# B&R Automation Studio project Kesim (part 5)

### CsvHandling.typ - Package data types
```iecst
(********************************************************************
 * COPYRIGHT -- Bernecker + Rainer
 ********************************************************************
 * Package: CSVHandling
 * File: CSVHandling.typ
 * Author: blanca-gutim
 * Created: December 04, 2012
 ********************************************************************
 * Data types of package CSVHandling
 ********************************************************************)
(**)
(*Enumeration to manage the state machine states*)

TYPE
	emu_CSVControl_State :
		(
		C_MS_CSV_FILE_HAND_INIT := 0, (*Init state*)
		C_MS_CSV_FILE_HAND_WAIT_CMD, (*Wait commad state -Standstill state*)
		C_MS_CSV_FILE_HAND_READ, (*Read CSV file state*)
		C_MS_CSV_FILE_HAND_GEN_FILE_NAME, (*Generate file name state*)
		C_MS_CSV_FILE_HAND_SEARCH_FILE, (*Search for the specified file name*)
		C_MS_CSV_FILE_HAND_WAIT_OVRW_OK, (*Wait overwrite confirmation state*)
		C_MS_CSV_FILE_HAND_SEARCH_VAR, (*Search the variables that are part of the CSV file state*)
		C_MS_CSV_FILE_HAND_WRITE, (*Write CSV file state*)
		C_MS_CSV_FILE_HAND_ERROR, (*General error state*)
		C_MS_CSV_FILE_HAND_ACK_ERROR, (*Acknowledge error state*)
		C_MS_CSV_FILE_HAND_NOERROR (*Error State - No error*)
		);
END_TYPE

(**)
(*========================================================================================================*)
(*CSV control interface type*)
(*========================================================================================================*)

TYPE
	CSV_Ctrl_typ : 	STRUCT
		In : CSV_Ctrl_In_typ; (*Inputs*)
		Out : CSV_Ctrl_Out_typ; (*Outputs*)
	END_STRUCT;
END_TYPE

(*========================================================================================================*)
(*CSV control: input sub-interface type*)
(*========================================================================================================*)

TYPE
	CSV_Ctrl_In_typ : 	STRUCT
		Cmd : CSV_Ctrl_In_Cmd_typ; (*Input commands*)
		Par : CSV_Ctrl_In_Par_typ; (*Input parameters *)
		Stat : CSV_Ctrl_In_Stat_typ; (*Input status*)
	END_STRUCT;
END_TYPE

(*CSV control: input commands sub-interface type*)

TYPE
	CSV_Ctrl_In_Cmd_typ : 	STRUCT
		ReadFile : BOOL; (*Read file command*)
		WriteFile : BOOL; (*Write file command*)
		OverwriteFile : BOOL; (*Overwrite file command*)
		NotOverwriteFile : BOOL; (*Do not overwrite file command*)
		ErrorAcknowledge : BOOL; (*Acknowledge error command*)
	END_STRUCT;
END_TYPE

(*CSV control: input parameters sub-interface type*)

TYPE
	CSV_Ctrl_In_Par_typ : 	STRUCT
		FileDeviceName : STRING[50]; (*File Device name*)
		FileName : STRING[255]; (*File name*)
		Path : STRING[255]; (*Path to the file*)
		Header : CSV_Ctrl_In_Par_Header_typ; (*Header input parameters substructure*)
	END_STRUCT;
END_TYPE

(*Header input parameters substructure*)

TYPE
	CSV_Ctrl_In_Par_Header_typ : 	STRUCT
		Enable : BOOL; (*Enable header in CSV file*)
		MachineNr : STRING[80]; (*Machine number*)
		Comment : STRING[80]; (*Header comment*)
		Version : STRING[80]; (*Version*)
	END_STRUCT;
END_TYPE

(*CSV control: input status sub-interface type*)

TYPE
	CSV_Ctrl_In_Stat_typ : 	STRUCT
		NOT_USED : BOOL;
	END_STRUCT;
END_TYPE

(*========================================================================================================*)
(*CSV control: output sub-interface type*)
(*========================================================================================================*)

TYPE
	CSV_Ctrl_Out_typ : 	STRUCT
		Cmd : CSV_Ctrl_Out_Cmd_typ; (*Output commands*)
		Par : CSV_Ctrl_Out_Par_typ; (*Output parameters *)
		Stat : CSV_Ctrl_Out_Stat_typ; (*Output status*)
	END_STRUCT;
END_TYPE

(*CSV control: output commands sub-interface type*)

TYPE
	CSV_Ctrl_Out_Cmd_typ : 	STRUCT
		NOT_USED : BOOL;
	END_STRUCT;
END_TYPE

(*CSV control: output parameters sub-interface type*)

TYPE
	CSV_Ctrl_Out_Par_typ : 	STRUCT
		NOT_USED : BOOL;
	END_STRUCT;
END_TYPE

(*CSV control: output status sub-interface type*)

TYPE
	CSV_Ctrl_Out_Stat_typ : 	STRUCT
		MainState : DINT; (*Main state in numeric format*)
		MainState_Text : STRING[32]; (*Main state in text format*)
		VariableNames : ARRAY[0..C_NR_VARIABLES_CSVFILE_MINUS1]OF STRING[30]; (*Names of the variables that are part of the CSV file*)
		CmdDone : CSV_Ctrl_In_Cmd_typ; (*Command done*)
		FileAlreadyExists : BOOL; (*Flag to show that the CSV file already exists (in write process)*)
		ReadyForCmd : BOOL; (*Variable to show that the program is ready to get a new command*)
(*		Error : Error_Type; (*Error information*)
	END_STRUCT;
END_TYPE
```

### CsvHandling.var - Package variables
```iecst
(********************************************************************
 * COPYRIGHT -- Bernecker + Rainer
 ********************************************************************
 * Package: RecipeHandling
 * File: CsvHandling.var
 * Author: blanca-gutim
 * Created: December 04, 2012
 ********************************************************************
 * Variables of package RecipeHandling
 ********************************************************************)
(**)
(*========================================================================================================*)
(*Program variables*)
(*========================================================================================================*)
VAR
	gCSV_Ctrl : CSV_Ctrl_typ; (*CSV control interface*)
END_VAR
```

### Program Logical/CuttingTable/RecipeHandling/CsvHandling/CSV_Ctrl (IEC) - CSV file control program

#### CSV_CtrlCyclic.st - Cyclic code
```iecst
(********************************************************************
 * COPYRIGHT -- Bernecker + Rainer
 ********************************************************************
 * PROGRAM: gCSV_Ctrl
 * File: gCSV_CtrlCyclic.st
 * Author: blanca-gutim
 * Created: December 06, 2012
 ********************************************************************
 * Implementation OF PROGRAM gCSV_Ctrl
 ********************************************************************)

PROGRAM _CYCLIC

	//Update inputs
	Action_Input;

	//====================================================================================================
	//
	//									MAIN STATE MACHINE
	//
	//====================================================================================================
	IF TON_Init.Q THEN
		TON_Init.IN := FALSE;
		//FUB execution
		Init_CSVHandling();

		//Check if the FUB is done
		IF (Init_CSVHandling.status = ERR_FUB_BUSY) THEN
			//The FUB is busy
		ELSE
			IF (Init_CSVHandling.status = ERR_OK) THEN
				//FUB executed successfully
			ELSE
				//Error -> Save information about error
				gCSV_Ctrl.Out.Stat.Error.Number		:= Init_CSVHandling.status;
				gCSV_Ctrl.Out.Stat.Error.Text.Line1	:= TaskName;
				gCSV_Ctrl.Out.Stat.Error.Text.Line2	:= StateStrings[MainState];
				ErrorState							:= MainState;
				MainState							:= C_MS_CSV_FILE_HAND_ERROR;
			END_IF
		END_IF
	END_IF;
	CASE MainState OF

		//============================================================================================
		C_MS_CSV_FILE_HAND_INIT:					//INITIALIZATION STATE
			//============================================================================================

			//Initialization done -> Go to Wait Command state
			MainState 			:= C_MS_CSV_FILE_HAND_WAIT_CMD;

		//============================================================================================
		C_MS_CSV_FILE_HAND_WAIT_CMD:				//STANDSTILL STATE
			//============================================================================================

			//WAIT FOR COMMANDS
			IF (gCSV_Ctrl.Out.Stat.ReadyForCmd = TRUE) THEN
				IF (gCSV_Ctrl.In.Cmd.ReadFile > OldInputs.Cmd.ReadFile) THEN
					//Go to Read CSV file state
					MainState			:= C_MS_CSV_FILE_HAND_READ;
				ELSIF (gCSV_Ctrl.In.Cmd.WriteFile > OldInputs.Cmd.WriteFile) THEN
					//Go to the first state when a file is written
					MainState			:= C_MS_CSV_FILE_HAND_SEARCH_FILE;
				ELSE
					//Stay in Wait Command state
					MainState 			:= C_MS_CSV_FILE_HAND_WAIT_CMD;
				END_IF
			END_IF

			//Update the output ReadyForCmd
			IF (MainState = C_MS_CSV_FILE_HAND_WAIT_CMD) THEN
				gCSV_Ctrl.Out.Stat.ReadyForCmd	:= TRUE;
			ELSE
				gCSV_Ctrl.Out.Stat.ReadyForCmd	:= FALSE;
			END_IF

		//============================================================================================
		C_MS_CSV_FILE_HAND_READ:				//READ CSV FILE
			//============================================================================================

			//FUB parameters
			ReadFile_CSVHandling.pDevice			:= ADR(gCSV_Ctrl.In.Par.FileDeviceName);
			ReadFile_CSVHandling.pPath				:= ADR(gCSV_Ctrl.In.Par.Path);
			ReadFile_CSVHandling.pFileName			:= ADR(gCSV_Ctrl.In.Par.FileName);
			ReadFile_CSVHandling.Separator			:= C_SEPARATOR;	//Check constant to see the ASCII code of the actual separator
			ReadFile_CSVHandling.No_DatatypControl	:= 1;
			ReadFile_CSVHandling.IgnoreError		:= 1;
			ReadFile_CSVHandling.Options			:= 0;

			//FUB execution
			ReadFile_CSVHandling();

			//Chec if the FUB is done
			IF (ReadFile_CSVHandling.status = ERR_FUB_BUSY) THEN
				//The FUB is busy
			ELSE
				IF (ReadFile_CSVHandling.status = ERR_OK) THEN
					//FUB executed successfully -> Go to wait command state
					MainState							:= C_MS_CSV_FILE_HAND_WAIT_CMD;
					//Set output status command done
					gCSV_Ctrl.Out.Stat.CmdDone.ReadFile	:= TRUE;
				ELSE
					//Error -> Save information about error
					gCSV_Ctrl.Out.Stat.Error.Number		:= ReadFile_CSVHandling.status;
					gCSV_Ctrl.Out.Stat.Error.Text.Line1	:= TaskName;
					gCSV_Ctrl.Out.Stat.Error.Text.Line2	:= StateStrings[MainState];
					ErrorState							:= MainState;
					MainState							:= C_MS_CSV_FILE_HAND_ERROR;
				END_IF
			END_IF

		//============================================================================================
		C_MS_CSV_FILE_HAND_SEARCH_FILE:				//SEARCH FOR THE SPECIFIED FILE NAME
			//============================================================================================

			//FUB parameters
			ToSearchFileName						:= gCSV_Ctrl.In.Par.Path;
			strcat(ADR(ToSearchFileName), ADR(gCSV_Ctrl.In.Par.FileName));
			SearchFileName_CSVHandling.pFileName	:= ADR(ToSearchFileName);
			SearchFileName_CSVHandling.pDevice		:= ADR(gCSV_Ctrl.In.Par.FileDeviceName);

			//FUB execution
			SearchFileName_CSVHandling();

			//Chec if the FUB is done
			IF (SearchFileName_CSVHandling.status = ERR_FUB_BUSY) THEN
				//The FUB is busy
			ELSE
				IF (SearchFileName_CSVHandling.status = FILE_NOT_FOUND) THEN
					//FUB executed successfully, and the file does not exist -> Go to search variables that are part of the CSV file
					MainState							:= C_MS_CSV_FILE_HAND_SEARCH_VAR;
				ELSIF  (SearchFileName_CSVHandling.status = FILE_FOUND) THEN
					//FUB executed successfully, the file already exists -> Set flag to show this state, wait for confirmation to overwrite the file
					gCSV_Ctrl.Out.Stat.FileAlreadyExists := TRUE;
					MainState							:= C_MS_CSV_FILE_HAND_WAIT_OVRW_OK;
				ELSE
					//Error -> Save information about error
					gCSV_Ctrl.Out.Stat.Error.Number		:= SearchFileName_CSVHandling.status;
					gCSV_Ctrl.Out.Stat.Error.Text.Line1	:= TaskName;
					gCSV_Ctrl.Out.Stat.Error.Text.Line2	:= StateStrings[MainState];
					ErrorState							:= MainState;
					MainState							:= C_MS_CSV_FILE_HAND_ERROR;
				END_IF
			END_IF

		//============================================================================================
		C_MS_CSV_FILE_HAND_WAIT_OVRW_OK:			//WAIT FOR USER CONFIRMATION TO OVERWRITE THE FILE
			//============================================================================================

			//Wait for an user command about the possibility of overwriting the file
			IF (gCSV_Ctrl.In.Cmd.OverwriteFile > OldInputs.Cmd.OverwriteFile) THEN
				//Reset flag and go to search variables that are part of the CSV file
				gCSV_Ctrl.Out.Stat.FileAlreadyExists 		:= FALSE;
				MainState									:= C_MS_CSV_FILE_HAND_SEARCH_VAR;
			ELSIF (gCSV_Ctrl.In.Cmd.NotOverwriteFile > OldInputs.Cmd.NotOverwriteFile) THEN
				//Set output status commands done, flag and go to wait command
				gCSV_Ctrl.Out.Stat.CmdDone.WriteFile			:= TRUE;
				gCSV_Ctrl.Out.Stat.CmdDone.NotOverwriteFile	:= TRUE;
				gCSV_Ctrl.Out.Stat.FileAlreadyExists 		:= FALSE;
				MainState									:= C_MS_CSV_FILE_HAND_WAIT_CMD;
			END_IF

		//============================================================================================
		C_MS_CSV_FILE_HAND_SEARCH_VAR:				//SEARCH VARIABLES THAT ARE PART OF THE CSV FILE
			//============================================================================================

			//FUB parameters
			Search_CSVHandling.pStructName		:= Init_CSVHandling.pStructName;
			Search_CSVHandling.NumOfStructs		:= Init_CSVHandling.NumOfStructs;
			Search_CSVHandling.pStructMem		:= Init_CSVHandling.pStructMem;
			Search_CSVHandling.MemLen			:= Init_CSVHandling.MemCounter;
			Search_CSVHandling.Options			:= 0;
			Search_CSVHandling.FullNameLenght	:= C_SHOW_VAR_NAME_OPTION;
			Search_CSVHandling.FileHeader		:= gCSV_Ctrl.In.Par.Header.Enable;
			Search_CSVHandling.Separator		:= C_SEPARATOR; //Check constants to see the ASCII code
			Search_CSVHandling.pMaschineNo		:= ADR(gCSV_Ctrl.In.Par.Header.MachineNr);
			Search_CSVHandling.pComment			:= ADR(gCSV_Ctrl.In.Par.Header.Comment);
			Search_CSVHandling.pVersion			:= ADR(gCSV_Ctrl.In.Par.Header.Version);

			//FUB execution
			Search_CSVHandling;

			//Chec if the FUB is done
			IF (Search_CSVHandling.status = ERR_FUB_BUSY) THEN
				//The FUB is busy
			ELSE
				IF (Search_CSVHandling.status = ERR_OK) THEN
					//FUB executed successfully -> Go to write CSV file
					MainState							:= C_MS_CSV_FILE_HAND_WRITE;
				ELSE
					//Error -> Save information about error
					gCSV_Ctrl.Out.Stat.Error.Number		:= Search_CSVHandling.status;
					gCSV_Ctrl.Out.Stat.Error.Text.Line1	:= TaskName;
					gCSV_Ctrl.Out.Stat.Error.Text.Line2	:= StateStrings[MainState];
					ErrorState							:= MainState;
					MainState							:= C_MS_CSV_FILE_HAND_ERROR;
				END_IF
			END_IF

		//============================================================================================
		C_MS_CSV_FILE_HAND_WRITE:				//WRITE THE CSV FILE
			//============================================================================================

			//FUB parameters
			WriteFile_CSVHandling.pFileName		:= ADR(gCSV_Ctrl.In.Par.FileName);
			WriteFile_CSVHandling.pDevice		:= ADR(gCSV_Ctrl.In.Par.FileDeviceName);
			WriteFile_CSVHandling.pPath			:= ADR(gCSV_Ctrl.In.Par.Path);
			WriteFile_CSVHandling.pStructMem	:= Init_CSVHandling.pStructMem;
			WriteFile_CSVHandling.MemLen		:= Search_CSVHandling.FileLen;
			WriteFile_CSVHandling.Mode			:= FILE_OW;

			//FUB execution
			WriteFile_CSVHandling;

			//Chec if the FUB is done
			IF (WriteFile_CSVHandling.status = ERR_FUB_BUSY) THEN
				//The FUB is busy
			ELSE
				IF (WriteFile_CSVHandling.status = ERR_OK) THEN
					//FUB executed successfully -> Go to wait command
					MainState									:= C_MS_CSV_FILE_HAND_WAIT_CMD;
					//Set output status command done
					gCSV_Ctrl.Out.Stat.CmdDone.WriteFile			:= TRUE;
					IF (gCSV_Ctrl.In.Cmd.OverwriteFile = TRUE) THEN
						gCSV_Ctrl.Out.Stat.CmdDone.OverwriteFile	:= TRUE;
					END_IF
				ELSE
					//Error -> Save information about error
					gCSV_Ctrl.Out.Stat.Error.Number				:= WriteFile_CSVHandling.status;
					gCSV_Ctrl.Out.Stat.Error.Text.Line1			:= TaskName;
					gCSV_Ctrl.Out.Stat.Error.Text.Line2			:= StateStrings[MainState];
					ErrorState									:= MainState;
					MainState									:= C_MS_CSV_FILE_HAND_ERROR;
				END_IF
			END_IF

		//============================================================================================
		C_MS_CSV_FILE_HAND_ERROR:				//ERROR HANDLING
			//============================================================================================

			//Wait for user acknowledge
			IF (gCSV_Ctrl.In.Cmd.ErrorAcknowledge > OldInputs.Cmd.ErrorAcknowledge) THEN
				//The user wants to acknowledge the error -> Next step: Go to Acknowledge Error State
				MainState 				:= C_MS_CSV_FILE_HAND_ACK_ERROR;
			END_IF

		//============================================================================================
		C_MS_CSV_FILE_HAND_ACK_ERROR:			//ACKNOWLEDGE ERROR
			//============================================================================================

			//Clear error information
			gCSV_Ctrl.Out.Stat.Error.Number				:= 0;
			memset(ADR(gCSV_Ctrl.Out.Stat.Error.Text), 0, SIZEOF(gCSV_Ctrl.Out.Stat.Error.Text));
			ErrorState									:= C_MS_CSV_FILE_HAND_NOERROR;
			MainState									:= C_MS_CSV_FILE_HAND_WAIT_CMD;
			//Error acknowledged
			gCSV_Ctrl.Out.Stat.CmdDone.ErrorAcknowledge	:= TRUE;
			//Acknowledge done -> Next step: Go to Init State
			MainState 									:= C_MS_CSV_FILE_HAND_INIT;

		ELSE

			//============================================================================================

			//The program sould not come here
			MainState 								:= C_MS_CSV_FILE_HAND_ERROR;
			gCSV_Ctrl.Out.Stat.Error.Number			:= 0;
			gCSV_Ctrl.Out.Stat.Error.Text.Line1		:= TaskName;
			gCSV_Ctrl.Out.Stat.Error.Text.Line2		:= 'Not defined state in state machine';
			ErrorState								:= MainState;
			MainState								:= C_MS_CSV_FILE_HAND_ERROR;

			//============================================================================================

	END_CASE

	TON_Init();
	//Update old inputs variable
	OldInputs	:= gCSV_Ctrl.In;

	//Update outputs
	Action_Output;

END_PROGRAM
```

#### CSV_CtrlInit.st - Initialization code
```iecst
(********************************************************************
 * COPYRIGHT -- Bernecker + Rainer
 ********************************************************************
 * Program: gCSV_Ctrl
 * File: gCSV_CtrlInit.st
 * Author: blanca-gutim
 * Created: December 06, 2012
 ********************************************************************
 * Implementation of program gCSV_Ctrl
 ********************************************************************)

PROGRAM _INIT

	//Init of task name
	TaskName	:= 'CSV_Ctrl';

	//Init of variable to get state names in text format
	StateStrings[C_MS_CSV_FILE_HAND_INIT]			:= 'C_MS_CSV_FILE_HAND_INIT';
	StateStrings[C_MS_CSV_FILE_HAND_WAIT_CMD]		:= 'C_MS_CSV_FILE_HAND_WAIT_CMD';
	StateStrings[C_MS_CSV_FILE_HAND_READ]			:= 'C_MS_CSV_FILE_HAND_READ';
	StateStrings[C_MS_CSV_FILE_HAND_GEN_FILE_NAME]	:= 'C_MS_CSV_FILE_HAND_GEN_FILE_NAME';
	StateStrings[C_MS_CSV_FILE_HAND_SEARCH_FILE]	:= 'C_MS_CSV_FILE_HAND_SEARCH_FILE';
	StateStrings[C_MS_CSV_FILE_HAND_WAIT_OVRW_OK]	:= 'C_MS_CSV_FILE_HAND_WAIT_OVRW_OK';
	StateStrings[C_MS_CSV_FILE_HAND_SEARCH_VAR]		:= 'C_MS_CSV_FILE_HAND_SEARCH_VAR';
	StateStrings[C_MS_CSV_FILE_HAND_WRITE]			:= 'C_MS_CSV_FILE_HAND_WRITE';
	StateStrings[C_MS_CSV_FILE_HAND_ERROR]			:= 'C_MS_CSV_FILE_HAND_ERROR';
	StateStrings[C_MS_CSV_FILE_HAND_ACK_ERROR]		:= 'C_MS_CSV_FILE_HAND_ACK_ERROR';
	StateStrings[C_MS_CSV_FILE_HAND_NOERROR]		:= 'C_MS_CSV_FILE_HAND_NOERROR';

	//****************************************************************************************************************
	//****************************************************************************************************************
	//THIS PART OF THE CODE MUST BE CONFIGURED FOR EACH APPLICATION
	//CHECK THE VALUE OF THE CONSTANT: C_NR_VARIABLES_CSVFILE_MINUS_1
	//DELETE THE VARIABLES AND STRUCTURES FOR TESTING: TestVar1 AND TestVar2
	//****************************************************************************************************************
	//****************************************************************************************************************
	//Init of the variables that are going to take part in the CSV file
	//Addresses of the names of the variables
	pVarNames[0] 	:= ADR('gParameters');
	//Sizes of the variables
	VarSizes[0]		:= SIZEOF(gParameters);
	//Show output information about the involved variables
	gCSV_Ctrl.Out.Stat.VariableNames[0] := 'gParameters';
	//****************************************************************************************************************
	//****************************************************************************************************************

	//Init of machine state and error information
	MainState 	:= C_MS_CSV_FILE_HAND_INIT;
	ErrorState	:= C_MS_CSV_FILE_HAND_NOERROR;

	//================================================================================================================
	//Calculate the necessary size of the memory to save the CSV-file on the compact flash and allocate the memory
	//================================================================================================================

	//FUB parameters
	Init_CSVHandling.pStructName	:= ADR(pVarNames);
	Init_CSVHandling.NumOfStructs	:= C_NR_VARIABLES_CSVFILE_MINUS1 + 1;
	Init_CSVHandling.FullNameLenght	:= C_SHOW_VAR_NAME_OPTION;
	Init_CSVHandling.Options		:= 0;

	TON_Init.PT := T#5S;
	TON_Init.IN := TRUE;

END_PROGRAM
```

#### CSV_Ctrl.var - Local variables
```iecst
(********************************************************************
 * COPYRIGHT -- Bernecker + Rainer
 ********************************************************************
 * Program: CSV_Ctrl
 * File: CSV_Ctrl.var
 * Author: blanca-gutim
 * Created: December 06, 2012
 ********************************************************************
 * Local variables of program CSV_Ctrl
 ********************************************************************)
(**)
(*================================================
Program variables
================================================*)
VAR
	TaskName : STRING[20]; (*Name of the actual task, used for error handling*)
	MainState : emu_CSVControl_State; (*Main state for the control of the state machine*)
	ErrorState : emu_CSVControl_State; (*Variable used to identify in wich state an error occurs*)
	OldInputs : CSV_Ctrl_In_typ; (*Variable used to detect edges in the inputs*)
	StateStrings : ARRAY[0..15] OF STRING[32]; (*Array with the names of the possible states (update if the number of states is increased)*)
	pVarNames : ARRAY[0..C_NR_VARIABLES_CSVFILE_MINUS1] OF UDINT; (*Addresses of the variables that are part of the CSV file*)
	VarSizes : ARRAY[0..C_NR_VARIABLES_CSVFILE_MINUS1] OF UDINT; (*Sizes of the variables that are part of the CSV file*)
	ToSearchFileName : STRING[255] := ''; (*File name to search by the FUB*)
END_VAR
(**)
(*================================================*)
(*Constants*)
(*================================================*)
(**)
(**)
(*===========================================================================================================================================================*)
(*FUB´S DECLARATION*)
(*===========================================================================================================================================================*)
VAR
	Init_CSVHandling : CSV_Init; (*Calculate the necessary size of the memory to save the CSV-file on the compact flash and allocate the memory*)
	ReadFile_CSVHandling : CSV_ReadFile; (*Read a CSV-file*)
	Search_CSVHandling : CSV_Search; (*Search the specified variable (structure) and create the completed CSV_File entries in the RAM*)
	SearchFileName_CSVHandling : SearchFileName; (*Searching for a file name*)
	WriteFile_CSVHandling : CSV_WriteFile; (*Create a CSV-File with the entries, which are created form CSV_Search() *)
	TON_Init : TON;
END_VAR
```

#### Actions.st
```iecst
(********************************************************************
 * COPYRIGHT -- Bernecker + Rainer
 ********************************************************************
 * Program: gRecipe_Ctrl
 * File: Actions.st
 * Author: blanca-gutim
 * Created: December 04, 2012
 ********************************************************************
 * Implementation of program gRecipe_Ctrl
 ********************************************************************)

(* Input actions *)
ACTION Action_Input:

	//Update inputs
	gCSV_Ctrl.In.Cmd		:= gRecipe_Ctrl.Out.Cmd.CsvHandling;
	gCSV_Ctrl.In.Par		:= gRecipe_Ctrl.Out.Par.CsvHandling;

END_ACTION

(* Output actions *)
ACTION Action_Output:

	//Update outputs, reset command done status
	gCSV_Ctrl.Out.Stat.CmdDone.ErrorAcknowledge		:= gCSV_Ctrl.Out.Stat.CmdDone.ErrorAcknowledge	AND gCSV_Ctrl.In.Cmd.ErrorAcknowledge;
	gCSV_Ctrl.Out.Stat.CmdDone.NotOverwriteFile		:= gCSV_Ctrl.Out.Stat.CmdDone.NotOverwriteFile	AND gCSV_Ctrl.In.Cmd.NotOverwriteFile;
	gCSV_Ctrl.Out.Stat.CmdDone.OverwriteFile		:= gCSV_Ctrl.Out.Stat.CmdDone.OverwriteFile		AND gCSV_Ctrl.In.Cmd.OverwriteFile;
	gCSV_Ctrl.Out.Stat.CmdDone.ReadFile				:= gCSV_Ctrl.Out.Stat.CmdDone.ReadFile			AND gCSV_Ctrl.In.Cmd.ReadFile;
	gCSV_Ctrl.Out.Stat.CmdDone.WriteFile			:= gCSV_Ctrl.Out.Stat.CmdDone.WriteFile			AND gCSV_Ctrl.In.Cmd.WriteFile;

	//Update output, get MainState and Error State in String and UDINT variables (for tracing and debuging)
	gCSV_Ctrl.Out.Stat.MainState					:= MainState;
	gCSV_Ctrl.Out.Stat.MainState_Text				:= StateStrings[MainState];

END_ACTION
```

### Package Logical/CuttingTable/RecipeHandling/FileHandling - File handling program

### FileHandling.typ - Package data types
```iecst
(********************************************************************
 * COPYRIGHT -- Bernecker + Rainer
 ********************************************************************
 * Package: FileHandling
 * File: FileHandling.typ
 * Author: blanca-gutim
 * Created: December 04, 2012
 ********************************************************************
 * Data types of package FileHandling
 ********************************************************************)
(**)
(*Enumeration to manage the state machine states*)

TYPE
	emu_FileControl_State :
		(
		C_MS_FILE_HAND_INIT := 0, (*Init state*)
		C_MS_FILE_HAND_WAIT_CMD, (*Wait commad state -Standstill state*)
		C_MS_FILE_HAND_LINK_FILE_DEV, (*Link file device state*)
		C_MS_FILE_HAND_GET_DEV_INFO, (*Get file device information*)
		C_MS_FILE_HAND_UNLINK_FILE_DEV, (*Unlink file device state*)
		C_MS_FILE_HAND_DELETE_FILE, (*Delete file satte*)
		C_MS_FILE_HAND_OPEN_DIR, (*Open directory state*)
		C_MS_FILE_HAND_CLOSE_DIR, (*Close directory state*)
		C_MS_FILE_HAND_READ_DIR, (*Read directory state*)
		C_MS_FILE_HAND_CREATE_DIR, (*Create directory state*)
		C_MS_FILE_HAND_ERROR, (*General error state*)
		C_MS_FILE_HAND_ACK_ERROR, (*Acknowledge error state*)
		C_MS_FILE_HAND_NOERROR (*Error State - No error*)
		);
END_TYPE

(**)
(*========================================================================================================*)
(*File control interface type*)
(*========================================================================================================*)

TYPE
	File_Ctrl_typ : 	STRUCT
		In : File_Ctrl_In_typ; (*Inputs *)
		Out : File_Ctrl_Out_typ; (*Outputs*)
	END_STRUCT;
END_TYPE

(*========================================================================================================*)
(*File control: input sub-interface type*)
(*========================================================================================================*)

TYPE
	File_Ctrl_In_typ : 	STRUCT
		Cmd : File_Ctrl_In_Cmd_typ; (*Input commands *)
		Par : File_Ctrl_In_Par_typ; (*Input parameters *)
		Stat : File_Ctrl_In_Stat_typ; (*Input status*)
	END_STRUCT;
END_TYPE

(*File control: input commands sub-interface type*)

TYPE
	File_Ctrl_In_Cmd_typ : 	STRUCT
		LinkFileDevice : BOOL; (*Links a file device*)
		GetFileDeviceInfo : BOOL; (*Get file device information*)
		UnlinkFileDevice : BOOL; (*Unlinks file device*)
		ReadDirectory : BOOL; (*Reads a directory*)
		DeleteFile : BOOL; (*Deletes a file*)
		ErrorAcknowledge : BOOL; (*Acknowledges an error*)
	END_STRUCT;
END_TYPE

(*File control: input parameters sub-interface type*)

TYPE
	File_Ctrl_In_Par_typ : 	STRUCT
		DeviceName : STRING[50]; (*File device name*)
		ParameterString : STRING[255]; (*Device parameter string*)
		FileName : STRING[255]; (*File name*)
		DirectoryName : STRING[255]; (*Directory name*)
	END_STRUCT;
END_TYPE

(*File control: input status sub-interface type*)

TYPE
	File_Ctrl_In_Stat_typ : 	STRUCT
		NOT_USED : BOOL;
	END_STRUCT;
END_TYPE

(*========================================================================================================*)
(*File control: output sub-interface type*)
(*========================================================================================================*)

TYPE
	File_Ctrl_Out_typ : 	STRUCT
		Cmd : File_Ctrl_Out_Cmd_typ; (*Output commands *)
		Par : File_Ctrl_Out_Par_typ; (*Output parameters *)
		Stat : File_Ctrl_Out_Stat_typ; (*Output status *)
	END_STRUCT;
END_TYPE

(*File control: output commands sub-interface type*)

TYPE
	File_Ctrl_Out_Cmd_typ : 	STRUCT
		NOT_USED : BOOL;
	END_STRUCT;
END_TYPE

(*File control: output parameters sub-interface type*)

TYPE
	File_Ctrl_Out_Par_typ : 	STRUCT
		NOT_USED : BOOL;
	END_STRUCT;
END_TYPE

(*File control: output status sub-interface type*)

TYPE
	File_Ctrl_Out_Stat_typ : 	STRUCT
		MainState : DINT; (*Main state in numeric format*)
		MainState_Text : STRING[32]; (*Main state in text format*)
(*		UsbInformation : ARRAY[0..C_USB_DEVICES_MAX_MINUS1]OF usbNode_typ; (*Information about connected USB devices*)
		CmdDone : File_Ctrl_In_Cmd_typ; (*Command done*)
		FileDeviceInfo : File_Ctrl_Out_Stat_DevInfo_typ; (*Output device information*)
		DirectoryInformation : File_Ctrl_Out_Stat_DirInfo_typ; (*Output directory information*)
		ReadyForCmd : BOOL; (*Variable to show that the program is ready to get a new command*)
(*		Error : Error_Type; (*Error information*)
	END_STRUCT;
END_TYPE

(*File control: output status realted to the device info sub-interface type*)

TYPE
	File_Ctrl_Out_Stat_DevInfo_typ : 	STRUCT  (*Output device information*)
		FileDeviceLinked : BOOL; (*A file device is linked*)
		Name : STRING[50]; (*File device name*)
		FileDeviceHandle : UDINT; (*Device handle*)
		FreeMem : UDINT; (*Free memory*)
		TotalMem : UDINT; (*Total memory*)
	END_STRUCT;
END_TYPE

(*File control: output status realted to the read directory info sub-interface type*)

TYPE
	File_Ctrl_Out_Stat_DirInfo_typ : 	STRUCT  (*Output file information*)
		NrFiles : UDINT; (*Number of files in the directory*)
		NrDirectories : UDINT; (*Number os subdirectories in the directory*)
		ElementsInfo : ARRAY[0..C_MAX_NR_ELEMENTS_IN_DIR_MINUS1]OF fiDIR_READ_EX_DATA; (*Information about the elements inside the directory*)
	END_STRUCT;
END_TYPE
```

### FileHandling.var - Package variables
```iecst
(********************************************************************
 * COPYRIGHT -- Bernecker + Rainer
 ********************************************************************
 * Package: RecipeHandling
 * File: FileHandling.var
 * Author: blanca-gutim
 * Created: December 04, 2012
 ********************************************************************
 * Variables of package RecipeHandling
 ********************************************************************)
(**)
(*========================================================================================================*)
(*Program variables*)
(*========================================================================================================*)
VAR
	gFile_Ctrl : File_Ctrl_typ := (0); (*File control interface*)
END_VAR
```

### Program Logical/CuttingTable/RecipeHandling/FileHandling/File_Ctrl (IEC) - File control program

#### File_CtrlCyclic.st - Cyclic code
```iecst
(********************************************************************
 * COPYRIGHT -- Bernecker + Rainer
 ********************************************************************
 * Program: gFile_Ctrl
 * File: gFile_CtrlCyclic.st
 * Author: blanca-gutim
 * Created: December 06, 2012
 ********************************************************************
 * Implementation of program gFile_Ctrl
 ********************************************************************)

 (********************************************************************
  * FORMAT OF FILE DEVICES STRING PARAMETERS
  *	CF: 		'/DEVICE=C:\\'
  *				-> The path of the directory that will be the file device is needed
  * USB:		'/DEVICE=IF4.ST1'
  *				-> The path of the directory that will be the file device is needed
  * FTP:		'/SIP=172.16.1.198 /SNAME=FTP_SERV1 /PROTOCOL=ftp /USER=max /PASSWORD=passw'
  *				-> Only the IP address of the FTP server is needed
  * NETWORK: 	'/PROTOCOL=cifs /SIP=192.168.90.121 /SHARE=ShareDir /USER=blanca-gutim /PASSWORD=passw /DOMAIN=BRATEGGE'
  *				-> The following requirements must be done to work with NETWORK file devices
  *					-> SIP=192.168.90.121 	= IP address of the system (PC for example) where the Shared Directory is located
  *					-> SHARE 				= Name of the Sagred folder in the network
  *					-> USER					= User name in the network (there must be a user defined in the network in order to have access to it)
  *					-> PASSWORD				= User password in the network (there must be a user defined in the network in order to have access to it)
  *					-> DOMAIN				= Name of the network Workgroup (it is possibel to check the name in "Windows Explorer -> Network section" in the left side of the screen)
  *					-> The Shared Directory in the network must be created in the source system and configured properly to permit access
  ********************************************************************)

PROGRAM _CYCLIC

	//Update inputs
	Action_Input;

	//====================================================================================================
	//
	//									MAIN STATE MACHINE
	//
	//====================================================================================================

	CASE MainState OF

		//============================================================================================
		C_MS_FILE_HAND_INIT:						//INITIALIZATION STATE
		//============================================================================================

			//The file handling task doesn´t need to perform any special action
			MainState 			:= C_MS_FILE_HAND_WAIT_CMD;

		//============================================================================================
		C_MS_FILE_HAND_WAIT_CMD:					//READY STATE
		//============================================================================================

			//WAIT FOR COMMANDS
			IF (gFile_Ctrl.Out.Stat.ReadyForCmd = TRUE) THEN
				IF (gFile_Ctrl.In.Cmd.LinkFileDevice > OldInputs.Cmd.LinkFileDevice) THEN
					//Go to Link File Device state
					MainState			:= C_MS_FILE_HAND_LINK_FILE_DEV;
				ELSIF (gFile_Ctrl.In.Cmd.GetFileDeviceInfo > OldInputs.Cmd.GetFileDeviceInfo) THEN
					//Go to Get File Device Information state
					MainState			:= C_MS_FILE_HAND_GET_DEV_INFO;
				ELSIF (gFile_Ctrl.In.Cmd.UnlinkFileDevice > OldInputs.Cmd.UnlinkFileDevice) THEN
					//Go to Unlink File Device state
					MainState			:= C_MS_FILE_HAND_UNLINK_FILE_DEV;
				ELSIF (gFile_Ctrl.In.Cmd.DeleteFile > OldInputs.Cmd.DeleteFile) THEN
					//Go to Delete File state
					MainState			:= C_MS_FILE_HAND_DELETE_FILE;
				ELSIF (gFile_Ctrl.In.Cmd.ReadDirectory > OldInputs.Cmd.ReadDirectory) THEN
					//Reset the memory area where the data is stored
					memset(ADR(gFile_Ctrl.Out.Stat.DirectoryInformation.ElementsInfo), 0, SIZEOF(gFile_Ctrl.Out.Stat.DirectoryInformation.ElementsInfo));
					//Go to Open Directory state
					MainState			:= C_MS_FILE_HAND_OPEN_DIR;
				ELSE
					//Stay in Wait Command state
					MainState 			:= C_MS_FILE_HAND_WAIT_CMD;
				END_IF
			END_IF

			//Update the output ReadyForCmd
			IF (MainState = C_MS_FILE_HAND_WAIT_CMD) THEN
				gFile_Ctrl.Out.Stat.ReadyForCmd	:= TRUE;
			ELSE
				gFile_Ctrl.Out.Stat.ReadyForCmd	:= FALSE;
			END_IF

		//============================================================================================
		C_MS_FILE_HAND_LINK_FILE_DEV:		//LINK FILE DEVICE
		//============================================================================================

			//Enable FUB
			DevLink_FileHandling.enable		:= TRUE;

			//Update FUB parameters
			DevLink_FileHandling.pDevice	:= ADR(gFile_Ctrl.In.Par.DeviceName);
			DevLink_FileHandling.pParam		:= ADR(gFile_Ctrl.In.Par.ParameterString);

			//FUB execution
			DevLink_FileHandling();

			//Wait for FUB execution
			IF (DevLink_FileHandling.status = ERR_FUB_BUSY) THEN
				//FUB busy
			ELSE
				//Check if the FUB execution is finished or there is an error
				IF (DevLink_FileHandling.status = ERR_OK) THEN
					//FUB executed successfully -> Save output information and go to Wait command state
					gFile_Ctrl.Out.Stat.FileDeviceInfo.FileDeviceLinked 	:= TRUE;
					gFile_Ctrl.Out.Stat.FileDeviceInfo.FileDeviceHandle	:= DevLink_FileHandling.handle;
					gFile_Ctrl.Out.Stat.FileDeviceInfo.Name				:= gFile_Ctrl.In.Par.DeviceName;
					MainState											:= C_MS_FILE_HAND_WAIT_CMD;
					//Set command done
					gFile_Ctrl.Out.Stat.CmdDone.LinkFileDevice			:= TRUE;
				ELSE
					//ERROR in FUB -> Save error information and go to Error State
					gFile_Ctrl.Out.Stat.Error.Number		:= UINT_TO_UDINT(DevLink_FileHandling.status);
					gFile_Ctrl.Out.Stat.Error.Text.Line1	:= TaskName;
					gFile_Ctrl.Out.Stat.Error.Text.Line2	:= StateStrings[MainState];
					ErrorState							:= MainState;
					MainState							:= C_MS_FILE_HAND_ERROR;
				END_IF
				//Reset enable FUB input
				DevLink_FileHandling.enable	:= FALSE;
			END_IF

		//============================================================================================
		C_MS_FILE_HAND_GET_DEV_INFO:		//GET FILE DEVICE INFORMATION
		//============================================================================================

			//Enable FUB
			DevMemInfo_FileHandling.enable		:= TRUE;

			//Update FUB parameters
			DevMemInfo_FileHandling.pDevice		:= ADR(gFile_Ctrl.Out.Stat.FileDeviceInfo.Name);

			//FUB execution
			DevMemInfo_FileHandling();

			//Wait for FUB execution
			IF (DevMemInfo_FileHandling.status = ERR_FUB_BUSY) THEN
				//FUB busy
			ELSE
				//Check if the FUB execution is finished or there is an error
				IF (DevMemInfo_FileHandling.status = ERR_OK) THEN
					//FUB executed successfully -> Save output information and go to Wait command state
					gFile_Ctrl.Out.Stat.FileDeviceInfo.FreeMem		:= DevMemInfo_FileHandling.freemem;
					gFile_Ctrl.Out.Stat.FileDeviceInfo.TotalMem		:= DevMemInfo_FileHandling.memsize;
					MainState										:= C_MS_FILE_HAND_WAIT_CMD;
					//Set command done
					gFile_Ctrl.Out.Stat.CmdDone.GetFileDeviceInfo	:= TRUE;
				ELSE
					//ERROR in FUB -> Save error information and go to Error State
					gFile_Ctrl.Out.Stat.Error.Number					:= UINT_TO_UDINT(DevMemInfo_FileHandling.status);
					gFile_Ctrl.Out.Stat.Error.Text.Line1				:= TaskName;
					gFile_Ctrl.Out.Stat.Error.Text.Line2				:= StateStrings[MainState];
					ErrorState										:= MainState;
					MainState										:= C_MS_FILE_HAND_ERROR;
				END_IF
				//Reset enable FUB input
				DevMemInfo_FileHandling.enable						:= FALSE;
			END_IF

		//============================================================================================
		C_MS_FILE_HAND_UNLINK_FILE_DEV:		//UNLINK FILE DEVICE
		//============================================================================================

			//Enable FUB
			DevUnlink_FileHandling.enable		:= TRUE;

			//Update FUB parameters
			DevUnlink_FileHandling.handle		:= gFile_Ctrl.Out.Stat.FileDeviceInfo.FileDeviceHandle;

			//FUB execution
			DevUnlink_FileHandling();

			//Wait for FUB execution
			IF (DevUnlink_FileHandling.status = ERR_FUB_BUSY) THEN
				//FUB busy
			ELSE
				//Check if the FUB execution is finished or there is an error
				IF (DevUnlink_FileHandling.status = ERR_OK) THEN
					//FUB executed successfully -> Save output information and go to Wait command state
					gFile_Ctrl.Out.Stat.FileDeviceInfo.FileDeviceLinked 	:= FALSE;
					gFile_Ctrl.Out.Stat.FileDeviceInfo.FileDeviceHandle	:= 0;
					gFile_Ctrl.Out.Stat.FileDeviceInfo.Name				:= '';
					gFile_Ctrl.Out.Stat.FileDeviceInfo.FreeMem			:= 0;
					gFile_Ctrl.Out.Stat.FileDeviceInfo.TotalMem			:= 0;
					MainState											:= C_MS_FILE_HAND_WAIT_CMD;
					//Set command done
					gFile_Ctrl.Out.Stat.CmdDone.UnlinkFileDevice			:= TRUE;
				ELSE
					//ERROR in FUB -> Save error information and go to Error State
					gFile_Ctrl.Out.Stat.Error.Number					:= UINT_TO_UDINT(DevUnlink_FileHandling.status);
					gFile_Ctrl.Out.Stat.Error.Text.Line1				:= TaskName;
					gFile_Ctrl.Out.Stat.Error.Text.Line2				:= StateStrings[MainState];
					ErrorState											:= MainState;
					MainState											:= C_MS_FILE_HAND_ERROR;
				END_IF
				//Reset enable FUB input
				DevUnlink_FileHandling.enable	:= FALSE;
			END_IF

		//============================================================================================
		C_MS_FILE_HAND_DELETE_FILE:			//DELETE FILE
		//============================================================================================

			//Enable FUB
			FileDelete_FileHandling.enable		:= TRUE;

			//Update FUB parameters
			FileDelete_FileHandling.pDevice		:= ADR(gFile_Ctrl.Out.Stat.FileDeviceInfo.Name);
			FileDelete_FileHandling.pName		:= ADR(gFile_Ctrl.In.Par.FileName);

			//FUB execution
			FileDelete_FileHandling();

			//Wait for FUB execution
			IF (FileDelete_FileHandling.status = ERR_FUB_BUSY) THEN
				//FUB busy
			ELSE
				//Check if the FUB execution is finished or there is an error
				IF (FileDelete_FileHandling.status = ERR_OK) THEN
					//FUB executed successfully -> Go to Wait command state
					MainState								:= C_MS_FILE_HAND_WAIT_CMD;
					//Set command done
					gFile_Ctrl.Out.Stat.CmdDone.DeleteFile	:= TRUE;
				ELSE
					//ERROR in FUB -> Save error information and go to Error State
					gFile_Ctrl.Out.Stat.Error.Number			:= UINT_TO_UDINT(FileDelete_FileHandling.status);
					gFile_Ctrl.Out.Stat.Error.Text.Line1		:= TaskName;
					gFile_Ctrl.Out.Stat.Error.Text.Line2		:= StateStrings[MainState];
					ErrorState								:= MainState;
					MainState								:= C_MS_FILE_HAND_ERROR;
				END_IF
				//Reset enable FUB input
				FileDelete_FileHandling.enable	:= FALSE;
			END_IF

		//============================================================================================
		C_MS_FILE_HAND_OPEN_DIR:			//OPEN DIRECTORY
		//============================================================================================

			//Enable FUB
			DirOpen_FileHandling.enable		:= TRUE;

			//Update parameters
			DirOpen_FileHandling.pDevice	:=	ADR(gFile_Ctrl.Out.Stat.FileDeviceInfo.Name);
			DirOpen_FileHandling.pName		:= 	ADR(gFile_Ctrl.In.Par.DirectoryName);

			//FUB execution
			DirOpen_FileHandling();

			//Wait for FUB execution
			IF (DirOpen_FileHandling.status = ERR_FUB_BUSY) THEN
				//FUB busy
			ELSE
				//Check if the FUB execution is finished or there is an error
				IF (DirOpen_FileHandling.status = ERR_OK) THEN
					//FUB executed successfully -> Go to Read Directory state
					MainState					:= C_MS_FILE_HAND_READ_DIR;
					//Reset index to count elements into the directory
					jj 							:= 0;
					//Reset output information about directory
					memset(ADR(gFile_Ctrl.Out.Stat.DirectoryInformation), 0, SIZEOF(gFile_Ctrl.Out.Stat.DirectoryInformation));
				ELSIF (DirOpen_FileHandling.status = fiERR_DIR_NOT_EXIST) THEN
					//The directory is not found, create it
					MainState					:= C_MS_FILE_HAND_CREATE_DIR;
				ELSE
					//ERROR in FUB -> Save error information and go to Error State
					gFile_Ctrl.Out.Stat.Error.Number			:= UINT_TO_UDINT(DirOpen_FileHandling.status);
					gFile_Ctrl.Out.Stat.Error.Text.Line1		:= TaskName;
					gFile_Ctrl.Out.Stat.Error.Text.Line2		:= StateStrings[MainState];
					ErrorState									:= MainState;
					MainState									:= C_MS_FILE_HAND_ERROR;
				END_IF
				//Reset enable FUB input
				DirOpen_FileHandling.enable	:= FALSE;
			END_IF

		//============================================================================================
		C_MS_FILE_HAND_CREATE_DIR:			//CREATE FILE
		//============================================================================================

			//Enable FUB
			DirCreate_FileHandling.enable		:= TRUE;

			//Update FUB parameters
			DirCreate_FileHandling.pDevice		:=	ADR(gFile_Ctrl.Out.Stat.FileDeviceInfo.Name);
			DirCreate_FileHandling.pName		:= 	ADR(gFile_Ctrl.In.Par.DirectoryName);

			//FUB execution
			DirCreate_FileHandling();

			//Wait for FUB execution
			IF (DirCreate_FileHandling.status = ERR_FUB_BUSY) THEN
				//FUB busy
			ELSE
				//Check if the FUB execution is finished or there is an error
				IF (DirCreate_FileHandling.status = ERR_OK) THEN
					//FUB executed successfully -> Go to Wait command state
					MainState									:= C_MS_FILE_HAND_OPEN_DIR;
				ELSE
					//ERROR in FUB -> Save error information and go to Error State
					gFile_Ctrl.Out.Stat.Error.Number			:= UINT_TO_UDINT(DirCreate_FileHandling.status);
					gFile_Ctrl.Out.Stat.Error.Text.Line1		:= TaskName;
					gFile_Ctrl.Out.Stat.Error.Text.Line2		:= StateStrings[MainState];
					ErrorState									:= MainState;
					MainState									:= C_MS_FILE_HAND_ERROR;
				END_IF
				//Reset enable FUB input
				DirCreate_FileHandling.enable	:= FALSE;
			END_IF

		//============================================================================================
		C_MS_FILE_HAND_READ_DIR:			//READ DIRECTORY
		//============================================================================================

			//Enable FUB
			DirReadEx_FileHandling.enable		:= TRUE;

			//FUB parameters
			DirReadEx_FileHandling.pData		:= ADR(gFile_Ctrl.Out.Stat.DirectoryInformation.ElementsInfo[jj]);
			DirReadEx_FileHandling.ident		:= DirOpen_FileHandling.ident;
			DirReadEx_FileHandling.data_len		:= SIZEOF(gFile_Ctrl.Out.Stat.DirectoryInformation.ElementsInfo[0]);

			//FUB execution
			DirReadEx_FileHandling();

            IF jj >= C_MAX_NR_ELEMENTS_IN_DIR_MINUS1 THEN
                gFile_Ctrl.Out.Stat.Error.Number		:= 99998;
	            gFile_Ctrl.Out.Stat.Error.Text.Line1	:= TaskName;
	            gFile_Ctrl.Out.Stat.Error.Text.Line2	:= 'Too many files in directory';
	            ErrorState								:= MainState;
	            MainState								:= C_MS_FILE_HAND_ERROR ;
            END_IF

			//Wait for FUB execution
			IF (DirReadEx_FileHandling.status = ERR_FUB_BUSY) THEN
				//FUB busy
			ELSE
				//Check if the FUB execution is finished or there is an error
				IF (DirReadEx_FileHandling.status = fiERR_NO_MORE_ENTRIES ) THEN
					//Save number of files and directories
					gFile_Ctrl.Out.Stat.DirectoryInformation.NrDirectories	:= 0;
					gFile_Ctrl.Out.Stat.DirectoryInformation.NrFiles			:= 0;
					//Save the information only when the directory is not empty
					IF (jj <> 0) THEN
						FOR kk := 0 TO (jj - 1) BY 1 DO
							IF (gFile_Ctrl.Out.Stat.DirectoryInformation.ElementsInfo[kk].Mode = fiFILE) THEN
								gFile_Ctrl.Out.Stat.DirectoryInformation.NrFiles 		:= gFile_Ctrl.Out.Stat.DirectoryInformation.NrFiles + 1;
							ELSIF (gFile_Ctrl.Out.Stat.DirectoryInformation.ElementsInfo[kk].Mode = fiDIRECTORY) THEN
								gFile_Ctrl.Out.Stat.DirectoryInformation.NrDirectories 	:= gFile_Ctrl.Out.Stat.DirectoryInformation.NrDirectories + 1;
							END_IF
						END_FOR
					END_IF
					//FUB executed successfully -> Go to Close Directory state
					MainState								:= C_MS_FILE_HAND_CLOSE_DIR;
				ELSIF (DirReadEx_FileHandling.status = ERR_OK) THEN
					//Increment index to save the information
					jj 										:= jj + 1;
				ELSE
					//ERROR in FUB -> Save error information and go to Error State
					gFile_Ctrl.Out.Stat.Error.Number			:= UINT_TO_UDINT(DirReadEx_FileHandling.status);
					gFile_Ctrl.Out.Stat.Error.Text.Line1		:= TaskName;
					gFile_Ctrl.Out.Stat.Error.Text.Line2		:= StateStrings[MainState];
					ErrorState								:= MainState;
					MainState								:= C_MS_FILE_HAND_ERROR;
				END_IF
				//Reset enable FUB input
				DirReadEx_FileHandling.enable	:= FALSE;
			END_IF

		//============================================================================================
		C_MS_FILE_HAND_CLOSE_DIR:			//CLOSE DIRECTORY
		//============================================================================================

			//Enable FUB
			DirClose_FileHandling.enable		:= TRUE;

			//Update FUB parameters
			DirClose_FileHandling.ident			:= DirOpen_FileHandling.ident;

			//FUB execution
			DirClose_FileHandling();

			//Wait for FUB execution
			IF (DirClose_FileHandling.status = ERR_FUB_BUSY) THEN
				//FUB busy
			ELSE
				//Check if the FUB execution is finished or there is an error
				IF (DirClose_FileHandling.status = ERR_OK) THEN
					//FUB executed successfully -> Go to Wait command state
					MainState									:= C_MS_FILE_HAND_WAIT_CMD;
					//Set command done
					gFile_Ctrl.Out.Stat.CmdDone.ReadDirectory	:= TRUE;
				ELSE
					//ERROR in FUB -> Save error information and go to Error State
					gFile_Ctrl.Out.Stat.Error.Number				:= UINT_TO_UDINT(DirClose_FileHandling.status);
					gFile_Ctrl.Out.Stat.Error.Text.Line1			:= TaskName;
					gFile_Ctrl.Out.Stat.Error.Text.Line2			:= StateStrings[MainState];
					ErrorState									:= MainState;
					MainState									:= C_MS_FILE_HAND_ERROR;
				END_IF
				//Reset enable FUB input
				DirClose_FileHandling.enable					:= FALSE;
			END_IF

		//============================================================================================
		C_MS_FILE_HAND_ERROR:				//ERROR HANDLING
		//============================================================================================

			//Wait for user acknowledge
			IF (gFile_Ctrl.In.Cmd.ErrorAcknowledge > OldInputs.Cmd.ErrorAcknowledge) THEN
				//The user wants to acknowledge the error -> Next step: Go to Acknowledge Error State
				MainState 			:= C_MS_FILE_HAND_ACK_ERROR;
			END_IF

		//============================================================================================
		C_MS_FILE_HAND_ACK_ERROR:			//ACKNOWLEDGE ERROR
		//============================================================================================

			//Clear error information
			gFile_Ctrl.Out.Stat.Error.Number				:= 0;
			memset(ADR(gFile_Ctrl.Out.Stat.Error.Text), 0, SIZEOF(gFile_Ctrl.Out.Stat.Error.Text));
			ErrorState									:= C_MS_FILE_HAND_NOERROR;
			MainState									:= C_MS_FILE_HAND_WAIT_CMD;
			//Error acknowledged
			gFile_Ctrl.Out.Stat.CmdDone.ErrorAcknowledge	:= TRUE;
			//Acknowledge done -> Next step: Go to Init State
			MainState 									:= C_MS_FILE_HAND_INIT;

		ELSE

			//============================================================================================

			//The program sould not come here
			MainState 								:= C_MS_FILE_HAND_ERROR;
			gFile_Ctrl.Out.Stat.Error.Number			:= 0;
			gFile_Ctrl.Out.Stat.Error.Text.Line1		:= TaskName;
			gFile_Ctrl.Out.Stat.Error.Text.Line2		:= 'Not defined state in state machine';
			ErrorState								:= MainState;
			MainState								:= C_MS_FILE_HAND_ERROR;

			//============================================================================================

	END_CASE

	//Update old inputs variable
	OldInputs	:= gFile_Ctrl.In;

	//Update outputs
	Action_Output;

END_PROGRAM
```

#### File_CtrlInit.st - Initialization code
```iecst
(********************************************************************
 * COPYRIGHT -- Bernecker + Rainer
 ********************************************************************
 * Program: gFile_Ctrl
 * File: gFile_CtrlInit.st
 * Author: blanca-gutim
 * Created: December 06, 2012
 ********************************************************************
 * Implementation of program gFile_Ctrl
 ********************************************************************)

PROGRAM _INIT

	//Init of task name
	TaskName	:= 'File_Ctrl';

	//Init of variables used to control state machines
	MainState	:= C_MS_FILE_HAND_INIT;
	ErrorState	:= C_MS_FILE_HAND_NOERROR;

	//Init of USB detection
	USBDetectionIF.in.Enable		:= TRUE;
	USBDetectionIF.out.Step			:= USB_GETNODELIST;

	//Init of variable to get state names in text format
	StateStrings[C_MS_FILE_HAND_INIT]				:= 'C_MS_FILE_HAND_INIT';
	StateStrings[C_MS_FILE_HAND_WAIT_CMD]			:= 'C_MS_FILE_HAND_WAIT_CMD';
	StateStrings[C_MS_FILE_HAND_LINK_FILE_DEV]		:= 'C_MS_FILE_HAND_LINK_FILE_DEV';
	StateStrings[C_MS_FILE_HAND_GET_DEV_INFO]		:= 'C_MS_FILE_HAND_GET_DEV_INFO';
	StateStrings[C_MS_FILE_HAND_UNLINK_FILE_DEV]	:= 'C_MS_FILE_HAND_UNLINK_FILE_DEV';
	StateStrings[C_MS_FILE_HAND_DELETE_FILE]		:= 'C_MS_FILE_HAND_DELETE_FILE';
	StateStrings[C_MS_FILE_HAND_OPEN_DIR]			:= 'C_MS_FILE_HAND_OPEN_DIR';
	StateStrings[C_MS_FILE_HAND_CLOSE_DIR]			:= 'C_MS_FILE_HAND_CLOSE_DIR';
	StateStrings[C_MS_FILE_HAND_READ_DIR]			:= 'C_MS_FILE_HAND_READ_DIR';
	StateStrings[C_MS_FILE_HAND_CREATE_DIR]			:= 'C_MS_FILE_HAND_CREATE_DIR';
	StateStrings[C_MS_FILE_HAND_ERROR]				:= 'C_MS_FILE_HAND_ERROR';
	StateStrings[C_MS_FILE_HAND_ACK_ERROR]			:= 'C_MS_FILE_HAND_ACK_ERROR';
	StateStrings[C_MS_FILE_HAND_NOERROR]			:= 'C_MS_FILE_HAND_NOERROR';

END_PROGRAM
```

#### File_Ctrl.typ - Local data types
```iecst
(********************************************************************
 * COPYRIGHT -- Bernecker + Rainer
 ********************************************************************
 * Program: File_Ctrl
 * File: File_Ctrl.typ
 * Author: blanca-gutim
 * Created: December 06, 2012
 ********************************************************************
 * Local data types of program File_Ctrl
 ********************************************************************)
(*======================================================================================================================================*)
(*USB DETECTION STEPS (CPU)*)
(*======================================================================================================================================*)

TYPE
	USB_STEP_type :
		(
		USB_GETNODELIST := 0, (*Create list of actives USB devices*)
		USB_SEARCHDEVICE1, (*Get device data from the USB device*)
		USB_SEARCHDEVICE2 (*Get device data from the USB device*)
		);
END_TYPE

(*======================================================================================================================================*)
(*USB DATA INTERFACE (CPU)*)
(*======================================================================================================================================*)
(*Interface for the USB detection*)

TYPE
	usb_detec_typ : 	STRUCT  (*Interface for the USB detection*)
		in : usb_detec_in_typ; (*Input sub-interface*)
		out : usb_detec_out_typ; (*Output sub-interface*)
	END_STRUCT;
END_TYPE

(*======================================================================================================================================*)
(*USB DATA INTERFACE: INPUTS*)
(*======================================================================================================================================*)
(*Output sub-interface*)

TYPE
	usb_detec_in_typ : 	STRUCT
		Enable : BOOL; (*Enable USB detection*)
	END_STRUCT;
END_TYPE

(*======================================================================================================================================*)
(*USB DATA INTERFACE: OUTPUTS*)
(*======================================================================================================================================*)
(*Output sub-interface*)

TYPE
	usb_detec_out_typ : 	STRUCT
		Step : USB_STEP_type; (*Output sub-interface*)
		NrUSBDetectedDevices : USINT; (*Number of USB devices detected*)
		DeviceInfo : ARRAY[0..C_USB_DEVICES_MAX_MINUS1]OF usbNode_typ; (*Structure with the information of the detected USB device*)
	END_STRUCT;
END_TYPE
```

#### File_Ctrl.var - Local variables
```iecst
(********************************************************************
 * COPYRIGHT -- Bernecker + Rainer
 ********************************************************************
 * Program: File_Ctrl
 * File: File_Ctrl.var
 * Author: blanca-gutim
 * Created: December 06, 2012
 ********************************************************************
 * Local variables of program File_Ctrl
 ********************************************************************)
(**)
(*================================================
Program variables
================================================*)
VAR
	TaskName : STRING[20]; (*Name of the actual task, used for error handling*)
	MainState : emu_FileControl_State; (*Main state for the control of the state machine*)
	ErrorState : emu_FileControl_State; (*Variable used to identify in wich state an error occurs*)
	kk : UDINT; (*Variable used as counter in FOR loops*)
	jj : UDINT; (*Variable used as counter in FOR loops*)
	ii : UDINT; (*Variable used as counter in FOR loops*)
	OldInputs : File_Ctrl_In_typ; (*Variable used to detect edges in the inputs*)
	StateStrings : ARRAY[0..15] OF STRING[32]; (*Array with the names of the possible states (update if the number of states is increased)*)
	usbNodeList : ARRAY[0..C_USB_DEVICES_MAX_MINUS1] OF UDINT; (*List of USB nodes*)
	USBDetectionIF : usb_detec_typ; (*Variable with the interface for the USB detection*)
END_VAR
(**)
(*===========================================================================================================================================================*)
(*FUB´S DECLARATION*)
(*===========================================================================================================================================================*)
VAR
	DevLink_FileHandling : DevLink; (*FUB: links file device*)
	DevMemInfo_FileHandling : DevMemInfo; (*FUB: gets information about the file device*)
	DevUnlink_FileHandling : DevUnlink; (*FUB: unlinks file devices*)
	DirClose_FileHandling : DirClose; (*FUB: closes a directory*)
	DirCreate_FileHandling : DirCreate; (*FUB: creates a directory*)
	DirOpen_FileHandling : DirOpen; (*FUB: opens a directory*)
	DirReadEx_FileHandling : DirReadEx; (*FUB: Reads the individual file or directory names in a directory*)
	FileDelete_FileHandling : FileDelete; (*FUB: deletes a file*)
	UsbNodeListGet_USBDetec : UsbNodeListGet; (*FUB: get list of USB nodes*)
	UsbNodeGet_USBDetec2 : UsbNodeGet; (*FUB: get information of an specific USB node*)
	UsbNodeGet_USBDetec1 : UsbNodeGet; (*FUB: get information of an specific USB node*)
END_VAR
```

#### Actions.st
```iecst
(********************************************************************
 * COPYRIGHT -- Bernecker + Rainer
 ********************************************************************
 * Program: gRecipe_Ctrl
 * File: Actions.st
 * Author: blanca-gutim
 * Created: December 04, 2012
 ********************************************************************
 * Implementation of program gRecipe_Ctrl
 ********************************************************************)

(* Input actions *)
ACTION Action_Input:

	//Update inputs
	gFile_Ctrl.In.Cmd		:= gRecipe_Ctrl.Out.Cmd.FileHandling;
	gFile_Ctrl.In.Par		:= gRecipe_Ctrl.Out.Par.FileHandling;

	//USB detection
	Action_USB_Detection;

END_ACTION

(* Output actions *)
ACTION Action_Output:

	//Update outputs, reset command done status
	gFile_Ctrl.Out.Stat.CmdDone.DeleteFile			:= gFile_Ctrl.Out.Stat.CmdDone.DeleteFile			AND gFile_Ctrl.In.Cmd.DeleteFile;
	gFile_Ctrl.Out.Stat.CmdDone.ErrorAcknowledge	:= gFile_Ctrl.Out.Stat.CmdDone.ErrorAcknowledge		AND gFile_Ctrl.In.Cmd.ErrorAcknowledge;
	gFile_Ctrl.Out.Stat.CmdDone.GetFileDeviceInfo	:= gFile_Ctrl.Out.Stat.CmdDone.GetFileDeviceInfo	AND gFile_Ctrl.In.Cmd.GetFileDeviceInfo;
	gFile_Ctrl.Out.Stat.CmdDone.LinkFileDevice		:= gFile_Ctrl.Out.Stat.CmdDone.LinkFileDevice		AND gFile_Ctrl.In.Cmd.LinkFileDevice;
	gFile_Ctrl.Out.Stat.CmdDone.ReadDirectory		:= gFile_Ctrl.Out.Stat.CmdDone.ReadDirectory		AND gFile_Ctrl.In.Cmd.ReadDirectory;
	gFile_Ctrl.Out.Stat.CmdDone.UnlinkFileDevice	:= gFile_Ctrl.Out.Stat.CmdDone.UnlinkFileDevice		AND gFile_Ctrl.In.Cmd.UnlinkFileDevice;

	//Update output, get MainState and Error State in String and UDINT variables (for tracing and debuging)
	gFile_Ctrl.Out.Stat.MainState					:= MainState;
	gFile_Ctrl.Out.Stat.MainState_Text				:= StateStrings[MainState];

	//Update output, USB devices information
	gFile_Ctrl.Out.Stat.UsbInformation[0]			:= USBDetectionIF.out.DeviceInfo[0];
	gFile_Ctrl.Out.Stat.UsbInformation[1]			:= USBDetectionIF.out.DeviceInfo[1];

END_ACTION

(* USB detection *)
ACTION Action_USB_Detection:

	//==================================================================================================================
	//STATE MACHINE FOR THE DETECTION OF THE USB DEVICES IN THE CPU
	//==================================================================================================================

	IF (USBDetectionIF.in.Enable = TRUE) THEN

		CASE (USBDetectionIF.out.Step) OF

			//==================================================================================================================
			USB_GETNODELIST:
			//==================================================================================================================

				UsbNodeListGet_USBDetec.enable					:= TRUE;
				UsbNodeListGet_USBDetec.pBuffer					:= ADR(usbNodeList[0]);
				UsbNodeListGet_USBDetec.bufferSize				:= SIZEOF(usbNodeList);
				UsbNodeListGet_USBDetec.filterInterfaceClass	:= asusb_CLASS_MASS_STORAGE;
				UsbNodeListGet_USBDetec.filterInterfaceSubClass	:= asusb_SUBCLASS_SCSI_COMMAND_SET;
				UsbNodeListGet_USBDetec();
				IF (UsbNodeListGet_USBDetec.status = ERR_OK) THEN
					//USB device found, get information from the device and get the number of detected USB devices
					USBDetectionIF.out.NrUSBDetectedDevices := 0;
					FOR ii := 1 TO C_USB_DEVICES_MAX_MINUS1 BY 1 DO
						IF (usbNodeList[ii] <> 0) THEN
							USBDetectionIF.out.NrUSBDetectedDevices := USBDetectionIF.out.NrUSBDetectedDevices + 1;
						END_IF
					END_FOR
					USBDetectionIF.out.Step:= DINT_TO_UINT(USB_SEARCHDEVICE1);
				ELSIF (UsbNodeListGet_USBDetec.status = asusbERR_USB_NOTFOUND) THEN
					//The USB is not found -> Clear structure with information
					memset(ADR(USBDetectionIF.out.DeviceInfo), 0, SIZEOF(USBDetectionIF.out.DeviceInfo));
					USBDetectionIF.out.NrUSBDetectedDevices := 0;
				ELSE
					IF ((UsbNodeListGet_USBDetec.status = asusbERR_BUFSIZE) OR (UsbNodeListGet_USBDetec.status = asusbERR_NULLPOINTER)) THEN
						//* Error Handling */
						gFile_Ctrl.Out.Stat.Error.Number		:= UINT_TO_UDINT(UsbNodeListGet_USBDetec.status);
						gFile_Ctrl.Out.Stat.Error.Text.Line1	:= TaskName;
						gFile_Ctrl.Out.Stat.Error.Text.Line2	:= 'USB_GETNODELIST';
						ErrorState							:= MainState;
						MainState							:= C_MS_FILE_HAND_ERROR;
					END_IF
				END_IF

			//==================================================================================================================
			USB_SEARCHDEVICE1:
			//==================================================================================================================

				UsbNodeGet_USBDetec1.enable		:= TRUE;
				UsbNodeGet_USBDetec1.nodeId		:= usbNodeList[0];
				UsbNodeGet_USBDetec1.pBuffer	:= ADR(USBDetectionIF.out.DeviceInfo[0]);
				UsbNodeGet_USBDetec1.bufferSize	:= SIZEOF(USBDetectionIF.out.DeviceInfo[0]);
				UsbNodeGet_USBDetec1();
				IF (UsbNodeGet_USBDetec1.status = ERR_OK) THEN
					//No errors -> Check for the other USB or get the list of USB again
					IF (USBDetectionIF.out.NrUSBDetectedDevices = 0) THEN
						USBDetectionIF.out.Step:= DINT_TO_UINT(USB_GETNODELIST);
						//Clear the information abot the second USB device
						memset(ADR(USBDetectionIF.out.DeviceInfo[1]), 0, SIZEOF(USBDetectionIF.out.DeviceInfo[1]));
					ELSE
						USBDetectionIF.out.Step:= DINT_TO_UINT(USB_SEARCHDEVICE2);
					END_IF
				ELSIF (UsbNodeGet_USBDetec1.status = asusbERR_USB_NOTFOUND) THEN
					//The USB is not found -> Clear structure with information and go to the previous step
					memset(ADR(USBDetectionIF.out.DeviceInfo[0]), 0, SIZEOF(USBDetectionIF.out.DeviceInfo[0]));
					USBDetectionIF.out.Step:= DINT_TO_UINT(USB_GETNODELIST);
				ELSE
					IF ((UsbNodeGet_USBDetec1.status = asusbERR_BUFSIZE) OR (UsbNodeGet_USBDetec1.status = asusbERR_NULLPOINTER)) THEN
						//* Error Handling */
						gFile_Ctrl.Out.Stat.Error.Number		:= UINT_TO_UDINT(UsbNodeGet_USBDetec1.status);
						gFile_Ctrl.Out.Stat.Error.Text.Line1	:= TaskName;
						gFile_Ctrl.Out.Stat.Error.Text.Line2	:= 'USB_SEARCHDEVICE1';
						ErrorState							:= MainState;
						MainState							:= C_MS_FILE_HAND_ERROR;
					END_IF
				END_IF

			//==================================================================================================================
			USB_SEARCHDEVICE2:
				//==================================================================================================================

				UsbNodeGet_USBDetec2.enable		:= TRUE;
				UsbNodeGet_USBDetec2.nodeId		:= usbNodeList[1];
				UsbNodeGet_USBDetec2.pBuffer	:= ADR(USBDetectionIF.out.DeviceInfo[1]);
				UsbNodeGet_USBDetec2.bufferSize	:= SIZEOF(USBDetectionIF.out.DeviceInfo[1]);
				UsbNodeGet_USBDetec2();
				IF (UsbNodeGet_USBDetec2.status = ERR_OK) THEN
					//No errors -> Get the list of USB again
					USBDetectionIF.out.Step:= DINT_TO_UINT(USB_GETNODELIST);
				ELSIF (UsbNodeGet_USBDetec2.status = asusbERR_USB_NOTFOUND) THEN
					//The USB is not found -> Clear structure with information and go to the previous step
					memset(ADR(USBDetectionIF.out.DeviceInfo[1]), 0, SIZEOF(USBDetectionIF.out.DeviceInfo[1]));
					USBDetectionIF.out.Step:= DINT_TO_UINT(USB_GETNODELIST);
				ELSE
					IF ((UsbNodeGet_USBDetec2.status = asusbERR_BUFSIZE) OR (UsbNodeGet_USBDetec2.status = asusbERR_NULLPOINTER)) THEN
						//* Error Handling */
						gFile_Ctrl.Out.Stat.Error.Number		:= UINT_TO_UDINT(UsbNodeGet_USBDetec2.status);
						gFile_Ctrl.Out.Stat.Error.Text.Line1	:= TaskName;
						gFile_Ctrl.Out.Stat.Error.Text.Line2	:= 'USB_SEARCHDEVICE2';
						ErrorState							:= MainState;
						MainState							:= C_MS_FILE_HAND_ERROR;
					END_IF
				END_IF

		END_CASE

	ELSE
		//Reset output information
		memset(ADR(USBDetectionIF.out), 0, SIZEOF(USBDetectionIF.out));

	END_IF

END_ACTION
```

- Visualisation Logical/mappView (not shown)

### Global.typ - not listed in the package file held
```iecst
TYPE
	gParameters_type : 	STRUCT
		MachineType : MachineTypes_Enm;
	END_STRUCT;
END_TYPE
```

### Parameters.typ - not listed in the package file held
```iecst
(********************************************************************
 * COPYRIGHT -- Bernecker + Rainer
 ********************************************************************
 * Package: CuttingTable
 * File: Parameter.typ
 * Author: blanca-gutim
 * Created: December 07, 2012
 ********************************************************************
 * Data types of package CuttingTable
 ********************************************************************)
(**)
(*========================================================================================================*)
(*Structure with machine parameters*)
(*========================================================================================================*)

TYPE
	gParameters_type : 	STRUCT
		BridgeStraight : BOOL; (*Command is taken from the HMI when the bridge straightness is set by the user*)
		MachineType : USINT; (*Machine type*)
		Options : Parameters_Options_typ;
		LengthParametes : LengthParametes_type; (*Length parameters*)
		DriverParameters : ARRAY[0..5]OF DriverParameters_type; (*Drive parameters*)
		PressParameters : PressParameters_type; (*Pressure parameters*)
(*		LoaderParameters : LoaderCtrl_In_Par_typ; (*Loader parameters*)
		Network : Recipe_Ctrl_In_Par_Net_typ; (*Network parameters*)
	END_STRUCT;
END_TYPE

(**)
(*========================================================================================================*)
(*Options*)
(*========================================================================================================*)

TYPE
	Parameters_Options_typ : 	STRUCT
		HW : Parameters_Options_HW_typ; (*Cutting table HW options*)
		SW : Parameters_Options_SW_typ; (*Cutting table SW options*)
	END_STRUCT;
	Parameters_Options_HW_Gantry_typ : 	STRUCT
		Active : BOOL;
		HoldingBrakes : BOOL;
		MultiturnEnc : BOOL;
	END_STRUCT;
	Parameters_Options_HW_typ : 	STRUCT
		LinearMotors_v1 : BOOL;
		LinearMotors_v2 : BOOL;
		NewLowE : BOOL; (*New version of the Low-E*)
		InkJet : {REDUND_UNREPLICABLE} BOOL; (*Inkjet printer exists in the machine instead of the old labeler system*)
		Labeler : BOOL;
		CAxisRev0 : BOOL; (*Revision xx-0 for the C axis [since it's a resolver, this should be known within the system so that the HW cfg is done accordingly]*)
		Gantry : Parameters_Options_HW_Gantry_typ;
		OCKMEnableTransferToBT : BOOL; (*Requested by the customer for one machine [14.05.2015].
The feature enables the glass transfer from the table to another machine in line. The process is the same with the YCKM_BREAKERs*)
	END_STRUCT;
	Parameters_Options_SW_typ : 	STRUCT
		TorqueDiffTimeout : REAL;
		TorqueDiffLimit : REAL;
		GanTorqMonTimeoutError : USINT; (*Option to treat the torque difference monitoring timeout as an error; by default it is treated as a warning*)
		NewGCodeRecipe : BOOL;
		GantryTorqueMonActive : BOOL; (*Option to activate the torque difference monitoring *)
		KeepBridgeEnabled : BOOL; (*Option keep the bridge axes enabled all the time*)
		AutoHwCfg : BOOL;
		AutoUserLogout : BOOL; (*Option to de/activate the automatic user logout functionality*)
		ManualOptimization : BOOL; (*Option to de/activate the manual optimization feature (since version  A3.54.0)*)
		LanguageEnable : ARRAY[0..9]OF BOOL; (*Enable the corresponding language to make it selectible on the HMI when the translations are there*)
	END_STRUCT;
END_TYPE

(**)
(*========================================================================================================*)
(*Length parameters*)
(*========================================================================================================*)

TYPE
	LengthParametes_type : 	STRUCT
		BAxisHomePos : REAL;
		BAxisMultiSetPos : REAL;
		YAxisMultiSetPos : REAL; (*Multiturn encoder home offset value for the Y axis [mm] / 0 when not applicable*)
		YAxisMultiHomeOffset : REAL; (*Set position for the multiturn encoder for the Y axis [mm] / 0 when not applicable*)
		MasterHomeOffset : REAL; (*Multiturn encder home offset value for master X axis [mm]*)
		MasterMultiSetPos : REAL; (*Set position of the multiturn encoder for the master*)
		SlaveHomeOffset : REAL; (*Multiturn encder home offset value for slave X2 axis [units]*)
		SlaveMultiSetPos : REAL; (*Set position of the multiturn encoder for the slave*)
		HeadUpTime : REAL; (*Time for the cutting head to move up [s]*)
		HeadDownTime : REAL; (*Time for the cutting head to move down [s]*)
		Low_eAboveTime : REAL; (*Time for the Low-E head to move up [s]*)
		Low_eBelowTime : REAL; (*Time for the Low-E head to move down [s]*)
		WaitPressureTime : REAL; (*Time to wait for the pressure reached [s]*)
		SquareForwardTime : REAL; (*Time to wait for the square forward movement [s]*)
		StretchingTime : REAL; (*Time to define how long the oil must be pumped when the machine starts operation [s] - NOT USED NOW*)
		X_GlassOriginPos : REAL; (*X distance between the Reference position and the Glass Origin position when the glass is placed without shift or rotation [mm]*)
		Y_GlassOriginPos : REAL; (*Y distance between the Reference position and the Glass Origin position when the glass is placed without shift or rotation [mm]*)
		C_GlassOriginPos : REAL; (*Offset between the cutting head and the glass (alignment) [°] - IT HAS TO BE MEASURED*)
		Y_GlassOriginPos_Right : REAL; (*Y distance between the Glass Origin position in the right side of the machine and the positive software limit in Y direction[mm] - ONLY IN FCL BIG SIZE MACHINES*)
		OffsetSpeed : REAL; (*Speed to move to Origin position [% prespect to maximum speed]*)
		X_AxisOffsetMachine : REAL; (*X offset between the cutting head and the laser sensor [mm]*)
		Y_AxisOffsetMachine : REAL; (*Y offset between the cutting head and the laser sensor [mm]*)
		Distance_Lowe_CuttingHead_X : REAL; (*X distance between cutting head and Low-E head [mm] *)
		Distance_Lowe_CuttingHead_Y : REAL; (*Y distance between cutting head and Low-E head [mm]*)
		X_HomeOffsetPos : REAL; (*X axis home offset [mm] - IT DEFINES THE REFERENCE POSITION, WHERE AXES ARE 0 units*)
		Y_HomeOffsetPos : REAL; (*Y axis home offset [mm] - IT DEFINES THE REFERENCE POSITION, WHERE AXES ARE 0 units*)
		C_HomeOffsetPos : REAL; (*C axis home offset [°] - IT DEFINES THE REFERENCE POSITION, WHERE AXES ARE 0 units*)
		ParkSpeed : REAL; (*Speed to move to Park position [% prespect to maximum speed]*)
		X3_Offset : REAL;
		X2_Offset : REAL;
		Y1_Offset : REAL;
		X_SafeLoadPosition : REAL; (*X axis position mandatory before loading*)
		MoveSafeLoadSpeed : REAL; (*Speed at which bridge will move to safe loading position*)
		Y_SafeLoadPosition : REAL; (*Y axis position mandatory before loading*)
		X_GlassTransferEndPosition : REAL; (*X axis, end position of transfer of the glass to breaking table*)
		Y_GlassTransferEndPosition : REAL; (*Y axis, end position of transfer of the glass to breaking table*)
		HomeSpeedTrigger : REAL;
		AutoSquaringSpeed : REAL; (*Auto squaring speed from the memory*)
		PushGlassSpeed : REAL; (*Speed at which glass should be transfered pushed after loading*)
		TransferSpeed : REAL; (*Speed at which glass should be transfered to breaking table*)
		StraightBridgeDelta : DINT; (*Defined by user, offset between ref pulses of X and X2 axes, having this parameter we can establish straigh position of bridge*)
		X_PushPositionEnd : REAL; (*Position when to finish glass pushing*)
		Y_PushPositionEnd : REAL; (*Position when to finish glass pushing*)
		Y_TransferPositionStart : REAL; (*Position when to start glass pushing/transfering*)
		X_TransferPositionStart : REAL; (*Position when to start glass pushing/transfering*)
		LabelApplyTime : REAL; (*Label application time*)
		InkJetPrintStroke : {REDUND_UNREPLICABLE} REAL; (*Stroke within which the inkjet should print*)
		InkJetPrintSpeed : {REDUND_UNREPLICABLE} REAL; (*Optimum speed at which the inkjet should perform the print (PLC will check the actual path speed of the CNC and trigger the print)*)
	END_STRUCT;
END_TYPE

(*========================================================================================================*)
(*Drive parameters*)
(*========================================================================================================*)

TYPE
	DriverParameters_type : 	STRUCT
		CntDir : USINT; (*Encoder counting direction*)
		DriveStep : REAL; (*Units needed for the motor to complete one turn [um] - THE SAME THAN units IN LOAD IN ACP INIT TABLE*)
		PositiveLimit : REAL; (*Positive software limit [mm] - THE SAME THAN IN LOAD IN ACP INIT TABLE*)
		NegativeLimit : REAL; (*Negative software limit [mm] - THE SAME THAN IN LOAD IN ACP INIT TABLE*)
		PID : DriverParameters_PID_type; (*PID parameters - THE SAME THAN IN CONTROLLER IN ACP INIT TABLE*)
	END_STRUCT;
END_TYPE

(*========================================================================================================*)
(*Drive PID parameters*)
(*========================================================================================================*)

TYPE
	DriverParameters_PID_type : 	STRUCT
		A0 : REAL;
		A1 : REAL;
		B0 : REAL;
		B1 : REAL;
		FilterType : UINT;
		Mode : USINT; (*Controller mode*)
		SpeedController : DriverParameters_PID_kv_tn_type; (*PID parameters for speed controller*)
		PositionController : DriverParameters_PID_kv_tn_type; (*PID parameters for position controller*)
		FeedForward : DriverParameters_FF_type; (*Feed forward related parameters*)
	END_STRUCT;
END_TYPE

(*========================================================================================================*)
(*Drive PID parameters: kn and tv*)
(*========================================================================================================*)

TYPE
	DriverParameters_PID_kv_tn_type : 	STRUCT
		kv : REAL; (*Proportional amplification*)
		tn : REAL; (*Integral action time [s]*)
	END_STRUCT;
END_TYPE

(*========================================================================================================*)
(*Drive Feed forward parameters*)
(*========================================================================================================*)

TYPE
	DriverParameters_FF_type : 	STRUCT
		Torque_Pos : REAL; (*Torque in positive direction [Nm]*)
		Torque_Neg : REAL; (*Torque in negative direction [Nm]*)
		Torque_Load : REAL; (*Load torque [Nm]*)
		Kv_Torque : REAL; (*Speed torque factor [Nms]*)
		Inertia : REAL; (*Mass moment of inertia [kgm˛]*)
	END_STRUCT;
END_TYPE

(*========================================================================================================*)
(*Pressure parameters*)
(*========================================================================================================*)

TYPE
	PressParameters_type : 	STRUCT
		PressureCalibration : REAL; (*Coefficient to convert pressure value in Analog Output*)
		PressureCoefficent : REAL; (*Indicates the pressure value set in Automatic Mode page*)
		HeadDownPress : REAL; (*Pressure when the cutting head is moving down [bar]*)
		VinylCutPressure : REAL; (*Pressure when the vynil cutting is done*)
		LoweDownPressure : REAL; (*Low-e down pressure - used only for the new low-e system *)
		GlassType : Press_Params_Glass_type; (*Parameters dependent on the glass type*)
	END_STRUCT;
END_TYPE

(*========================================================================================================*)
(*Pressure parameters that are dependent on the glass type*)
(*========================================================================================================*)

TYPE
	Press_Params_Glass_type : 	STRUCT
		T2 : Glass_PressureType; (*Glass thickness equal to 2 mm*)
		T3 : Glass_PressureType; (*Glass thickness equal to 3 mm*)
		T4 : Glass_PressureType; (*Glass thickness equal to 4 mm*)
		T5 : Glass_PressureType; (*Glass thickness equal to 5 mm*)
		T6 : Glass_PressureType; (*Glass thickness equal to 6 mm*)
		T8 : Glass_PressureType; (*Glass thickness equal to 8 mm*)
		T10 : Glass_PressureType; (*Glass thickness equal to 10 mm*)
		T12 : Glass_PressureType; (*Glass thickness equal to 12 mm*)
		T15 : Glass_PressureType; (*Glass thickness equal to 15 mm*)
		T19 : Glass_PressureType; (*Glass thickness equal to 19 mm*)
	END_STRUCT;
END_TYPE

(*========================================================================================================*)
(*Pressure parameters that are dependent on the glass type*)
(*========================================================================================================*)

TYPE
	Glass_PressureType : 	STRUCT
		MFunctionStart : UINT; (*Value of the fist M-Function used for this pressure values*)
		Pressure : ARRAY[0..5]OF REAL; (*Set pressure for different kinds of cut [bar]*)
	END_STRUCT;
END_TYPE
```

### Global.var - not listed in the package file held
```iecst
VAR
	FirstVariable : USINT;
	gParameters : USINT;
END_VAR
```

### Parameters.var - not listed in the package file held
```iecst
(********************************************************************
 * COPYRIGHT -- Bernecker + Rainer
 ********************************************************************
 * Package: MachineManager
 * File: MachineManager.var
 * Author: blanca-gutim
 * Created: December 04, 2012
 ********************************************************************
 * Variables of package MachineManager
 ********************************************************************)
(**)
VAR CONSTANT
	FCM : USINT := 0;
	FCL : USINT := 1;
	OCKM : USINT := 2;
	YCKM : USINT := 3;
	YCKM_BREAKER : USINT := 4;
END_VAR
(*========================================================================================================*)
(*Cutting table parameters structure*)
(*========================================================================================================*)
VAR RETAIN
	gOldOffset : REAL := 0.0; (*Previous homing offset for th C axis*)
	gParameters : gParameters_type; (*Cutting table parametesr structure*)
	gTotalCounter : UDINT; (*Total counter variable*)
	gDailyCounter : UDINT; (*Daily counter variable*)
	gSpeedRate : REAL; (*Speed rate variable*)
	gPressureRate : REAL; (*Pressure variable*)
	gDay : DATE; (*Variable with day information*)
	gMaxWorkCycles : UDINT; (*Maximum number of cycles until the machine is locked*)
END_VAR
VAR
	gFactorySettings : gParameters_type; (*Structure with the factory settings*)
END_VAR
```

### Constants.var
```iecst
(********************************************************************
 * COPYRIGHT --  B&R Industrial Automation GmbH
 *******************************************************************
 * Task: AlarmX
 * Author: kay3a
 * Created: October 2, 2024/3:55 PM
 ********************************************************************)
(**)
(**** Max Single Alarm Constant*)
VAR CONSTANT
	LC_MAX_SNIPPET_ALARM_INDEX : UDINT := 25; (**** Olabilecek maksimum single alarm sayisi*)
END_VAR
(**)
(**)
(**)
(**)
(**** Alarm Category Constants*)
VAR CONSTANT
	LC_ALARM_Category0_Abort : USINT := 0;
	LC_ALARM_Category1_Stop : USINT := 1;
	LC_ALARM_Category2_Pause : USINT := 2;
	LC_ALARM_Category3_Info : USINT := 3;
	LC_MAX_ALARM_CATEGORY_INDEX : UDINT := 3; (**** Olabilecek maksimum single alarm sayisi*)
END_VAR
```

### Program Logical/Infastructure/UserXMgr

#### Types.typ
```iecst
(********************************************************************
 * COPYRIGHT --  B&R Industrial Automation GmbH
 *******************************************************************
 * Task: UserX
 * Author: kay3a
 * Created: October 3, 2024/4:58 PM
 ********************************************************************)
(**)
(**** Local Type*)

TYPE
	Loc_typ : 	STRUCT
		FB : Loc_FB_typ; (**** Local FB ler*)
		Cmd : Loc_Cmd_typ; (**** Komutlar*)
		Status : Loc_Status_typ; (**** Durumlar*)
		Par : Loc_Par_typ;
	END_STRUCT;
END_TYPE

(**)
(**** Local FB Type*)

TYPE
	Loc_FB_typ : 	STRUCT  (**** Local FB Type*)
		DirRead : FbDirRead;
		DirCreate : FbDirCreate; (**** UserX export/import file dosyalarini tuttmak için.*)
		UserXLogin : MpUserXLogin;
		UserXManagerUI : MpUserXManagerUI;
		UserXLoginUI : MpUserXLoginUI;
	END_STRUCT;
END_TYPE

(**)
(**** Local Cmd Type*)

TYPE
	Loc_Cmd_typ : 	STRUCT  (**** Local Cmd Type*)
		Export : BOOL;
		ConfirmOverwrite : BOOL;
	END_STRUCT;
END_TYPE

(**)
(**** Local Status Type*)

TYPE
	Loc_Status_typ : 	STRUCT  (**** Local Status Type*)
		FileDuplicate : BOOL;
		ExportComplete : BOOL;
		UserExportDisplayed : BOOL;
		UserXHmiState : HmiStateEnum;
		LastMgrConnectStatus : MpUserXUIStatusEnum;
	END_STRUCT;
END_TYPE

(**)
(**** Local Parmaeter Type*)

TYPE
	Loc_Par_typ : 	STRUCT  (**** Local Parmaeter Type*)
		UserXLoginUIConnect : MpUserXLoginUIConnectType;
		UserXMgrUIConnect : MpUserXMgrUIConnectType;
	END_STRUCT;
END_TYPE

(**)
(**)
(**)
(**)
(*Enumerations*)

TYPE
	HmiStateEnum :
		( (*State enumeration for HMI interaction*)
		USERX_START := 0,
		USERX_WAIT_FOR_DIALOG := 1,
		USERX_SET_RESPONSE := 2,
		USERX_CONFIRM_RESPONSE := 3,
		USERX_NEW_EXPORT := 4,
		USERX_FINISH := 5
		);
END_TYPE
```

#### HMIAction.st
```iecst
(********************************************************************
 * COPYRIGHT --  B&R Industrial Automation GmbH
 ********************************************************************
 * Task: UserX
 * Author: kay3a
 * Created: October 3, 2024/4:59 PM
 ********************************************************************
 * Description:
 ********************************************************************)
//==============================================================================
ACTION HMIAction:

	CASE Loc.Status.UserXHmiState OF
		USERX_START:
			IF NOT Loc.Par.UserXMgrUIConnect.Import.ShowDialog THEN
				Loc.Par.UserXMgrUIConnect.Import.ShowDialog := TRUE;
			ELSE
				Loc.Status.UserXHmiState := USERX_WAIT_FOR_DIALOG;
			END_IF
		USERX_WAIT_FOR_DIALOG:
			Loc.Par.UserXMgrUIConnect.Import.ShowDialog := FALSE;
			Loc.Status.UserXHmiState := USERX_SET_RESPONSE;
		USERX_SET_RESPONSE:
			IF NOT(Loc.Par.UserXMgrUIConnect.Status = mpUSERX_UI_STATUS_IDLE) THEN
				Loc.Par.UserXMgrUIConnect.Import.Dialog.Cancel := TRUE;
			ELSE
				Loc.Par.UserXMgrUIConnect.Import.Dialog.Cancel := FALSE;
				Loc.Status.UserXHmiState := USERX_CONFIRM_RESPONSE;
			END_IF
		USERX_CONFIRM_RESPONSE:
			IF Loc.Par.UserXMgrUIConnect.Status = mpUSERX_UI_STATUS_WAIT_DLG THEN
				Loc.Status.UserXHmiState := USERX_START;
			ELSE
				Loc.Status.UserXHmiState := USERX_FINISH;
			END_IF
		USERX_NEW_EXPORT:
			IF NOT Loc.Par.UserXMgrUIConnect.Export.ShowDialog AND Loc.Par.UserXMgrUIConnect.Status = mpUSERX_UI_STATUS_IDLE THEN
				Loc.Status.UserXHmiState := USERX_START;
			END_IF
		USERX_FINISH:

	END_CASE
	// If new updates are made via export execute a check
	IF Loc.Par.UserXMgrUIConnect.Export.ShowDialog THEN
		Loc.Status.UserXHmiState := USERX_NEW_EXPORT;
	END_IF

	//Duplicate file checks
	IF EDGEPOS(Loc.Par.UserXMgrUIConnect.Status = mpUSERX_UI_STATUS_WAIT_DLG AND Loc.Par.UserXMgrUIConnect.Export.Dialog.LayerStatus = 0) OR
		EDGEPOS(Loc.Par.UserXMgrUIConnect.Status = mpUSERX_UI_STATUS_WAIT_DLG AND Loc.Par.UserXMgrUIConnect.Import.Dialog.LayerStatus = 0) THEN
		Loc.FB.DirRead.Execute := TRUE;
	END_IF;
	Loc.FB.DirRead.Parameters.DeviceName := Loc.FB.UserXManagerUI.UISetup.FileDevice;
	Loc.FB.DirRead.Enable := TRUE;
	IF Loc.FB.DirRead.CommandDone THEN
		Loc.FB.DirRead.Execute := FALSE;
	END_IF;
	Loc.FB.DirRead();
	Loc.Status.FileDuplicate := FALSE;
	FOR i := 0 TO 19 (*((SIZEOF(Loc.FB.DirRead.ListedFile)/SIZEOF(Loc.FB.DirRead.ListedFile[0])) - 1)*) DO
		temp := Loc.Par.UserXMgrUIConnect.Export.Dialog.FileName;
		brsstrcat(ADR(temp),ADR('.usr'));
		IF (temp = Loc.FB.DirRead.ListedFile[i]) THEN
			Loc.Status.FileDuplicate := Loc.Cmd.Export;
		END_IF;
	END_FOR;

	IF Loc.Status.FileDuplicate AND (Loc.Cmd.ConfirmOverwrite) THEN
		Loc.Par.UserXMgrUIConnect.Export.Dialog.Confirm := TRUE;
		Loc.Cmd.Export := FALSE;
		Loc.Cmd.ConfirmOverwrite := FALSE;
	ELSIF NOT Loc.Status.FileDuplicate AND Loc.Cmd.Export THEN
		Loc.Par.UserXMgrUIConnect.Export.Dialog.Confirm := TRUE;
		Loc.Cmd.Export := FALSE;
	END_IF

	// Export confirmation pop-up handling
	IF EDGENEG(Loc.Status.UserXHmiState = USERX_NEW_EXPORT) THEN
		IF (Loc.Status.LastMgrConnectStatus = mpUSERX_UI_STATUS_EXECUTE) AND (Loc.Par.UserXMgrUIConnect.Status = mpUSERX_UI_STATUS_IDLE) THEN
			Loc.Status.ExportComplete := TRUE;
		END_IF;
	END_IF;
	IF Loc.Status.UserExportDisplayed THEN
		Loc.Status.ExportComplete := FALSE;
		Loc.Status.UserExportDisplayed := FALSE;
		Loc.Par.UserXMgrUIConnect.Export.Dialog.Confirm := FALSE;
	END_IF

END_ACTION
//==============================================================================
```

### Program Logical/Program

#### Cyclic.st
```iecst
PROGRAM _CYCLIC
	(* Insert code here *)
	New_Variable := New_Variable +1;

	(* Bismillah*)
END_PROGRAM
```

### Program Logical/Source/CncCtrl (IEC)

#### Types.typ
```iecst
(********************************************************************
 * COPYRIGHT --  B&R Industrial Automation GmbH
 *******************************************************************
 * Task: MAIN
 * Author: kay3a
 * Created: October 16, 2024/11:08 AM
 ********************************************************************)

TYPE
	Loc_typ : 	STRUCT  (**** Local Type*)
		FB : Loc_FB_typ; (**** Local FB Type*)
		Par : Loc_Par_typ;
		Cmd : Loc_Cmd_typ; (**** Local Command Type*)
		Status : Loc_Status_typ; (**** Local Status Type*)
	END_STRUCT;
END_TYPE

(**)
(**** Local FB Type*)

TYPE
	Loc_FB_typ : 	STRUCT  (**** Local FB Type*)
		PML : MpPackMLModule; (**** PML Function Block*)
		Cnc3Axis : MpCnc3Axis; (**** CNC FB*)
		DirCreate : FbDirCreate; (**** CNC Direction create*)
		FileCreate : FbFileCreate; (**** CNC File create*)
	END_STRUCT;
END_TYPE

(**)
(**** Local Par Type*)

TYPE
	Loc_Par_typ : 	STRUCT  (**** Local Par Type*)
		PML : MpPackMLModuleParType; (**** PML Parameters*)
		Cnc3Axis : MpCnc3AxisParType;
	END_STRUCT;
END_TYPE

(**)
(**** Local Cmd Type*)

TYPE
	Loc_Cmd_typ : 	STRUCT  (**** Local Cmd Type*)
		New_Member : USINT;
	END_STRUCT;
END_TYPE

(**)
(**** Local Status Type*)

TYPE
	Loc_Status_typ : 	STRUCT  (**** Local Status Type*)
		New_Member : USINT;
	END_STRUCT;
END_TYPE

(**)
```
